// Pulses HOME and waits for the configured home-position feedback.
// Loss of bReady returns the FB to Idle without confirming completion.

FUNCTION_BLOCK FB_FanucHoming

VAR_INPUT
	bStart			: BOOL; // Rising edge starts homing while Idle and bReady; FALSE clears the FB error.
	bReady			: BOOL; // Enable permissive from FB_FanucEnable; must remain TRUE throughout the sequence.
	tHomingTimeout	: TIME := T#30S; // Maximum wait for bAt_Home = TRUE after the HOME pulse completes.
	stStatus		: ST_FanucStatus; // Live robot-status signals from FB_FanucStatus.
END_VAR

VAR_IN_OUT
	stControl	: ST_FanucControl; // Shared FANUC control structure; this FB writes Home only.
END_VAR

VAR_OUTPUT
	bBusy	: BOOL; // TRUE while in RequestHome or WaitComplete.
	bDone	: BOOL; // TRUE for one PLC scan when bAt_Home is TRUE in WaitComplete.
	bError	: BOOL; // TRUE in Error after a homing timeout or invalid state; cleared by bStart = FALSE.
	eState	: E_FanucHomingState; // Current state exposed for diagnostics and HMI.
END_VAR

VAR
	eCurrentState		: E_FanucHomingState := E_FanucHomingState.Idle; // Internal state used by the sequence.
	rtStart				: R_TRIG; // Detects the FALSE-to-TRUE transition of bStart.
	tonHomePulse		: TON; // Measures the HOME pulse duration in RequestHome.
	tonHomingTimeout	: TON; // Measures the wait for bAt_Home = TRUE in WaitComplete.
END_VAR

VAR CONSTANT
	tHomePulse	: TIME := T#200MS; // Requested duration of the HOME output pulse on UI[7].
END_VAR

(*
    FB_FanucHoming

    Purpose
    -------
    Controls the FANUC homing sequence and generates the HOME (UI[7])
    command used to trigger the configured homing macro or program.


    Homing sequence
    ---------------

        Idle
          |
          | bStart rising edge
          | + bReady
          v
        RequestHome
          |
          | HOME asserted for tHomePulse
          v
        WaitComplete
          |
          | bAt_Home = TRUE
          v
        Done
          |
          | one PLC scan
          v
        Idle


    Start behavior
    --------------
    bStart is treated as a momentary command.

    The R_TRIG detects the actual external FALSE -> TRUE transition:

        rtStart(CLK := bStart);

    The edge is accepted only when:

        bReady = TRUE
        AND
        eCurrentState = Idle

    A Start edge occurring while the robot is not Ready is ignored.

    If bStart goes TRUE before bReady becomes TRUE and remains TRUE,
    becoming Ready must NOT automatically start homing.

    bStart must first return FALSE and then receive a new rising edge.


    HOME pulse
    ----------
    RequestHome represents the HOME command pulse state.

    While RequestHome is active:

        stControl.Home = TRUE

    The HOME signal remains asserted for:

        tHomePulse

    After the pulse completes, the FB transitions to WaitComplete.


    Homing completion
    -----------------
    While in WaitComplete, the FB waits for:

        stStatus.bAt_Home = TRUE

    Once confirmed, the FB transitions to Done.

    bDone is TRUE for one PLC scan before the state returns to Idle.


    Ready interlock
    ---------------
    Homing may only start while:

        bReady = TRUE

    If bReady becomes FALSE during RequestHome or WaitComplete,
    the FB stops considering the homing sequence valid and returns
    to Idle.

    Returning this FB to Idle does not necessarily cancel a FANUC
    program or macro that has already started. Actual robot stopping
    behavior is controlled by the FANUC controller and its other UOP
    control inputs.


    Timeout
    -------
    While in WaitComplete, tonHomingTimeout runs for:

        tHomingTimeout

    If bAt_Home is not confirmed before the timeout expires,
    the FB transitions to Error.


    Error reset
    -----------
    To leave Error:

        bStart := FALSE

    The FB then returns to Idle.

    A new FALSE -> TRUE edge of bStart is required before another
    homing sequence can begin.


    FANUC prerequisites
    -------------------
    - HOME (UI[7]) must be configured to trigger the required
      homing macro or program.

    - stStatus.bAt_Home must represent the FANUC home-position
      feedback used by the application.


    Usage
    -----
    - Call this FB every PLC cycle.

    - Wire bReady from:

          FB_FanucEnable.bReady

    - Pass the same stControl instance used by the other FANUC
      command FBs and by FB_FanucControl.

    - Generate a rising edge on bStart to request homing.

    - Monitor:

          bBusy
          bDone
          bError
          eState
*)

// Start edge detection
// ============================================================================
//
// Detect the real external FALSE -> TRUE transition.
// Do not gate R_TRIG with bReady.
//
rtStart(CLK := bStart);

// State machine
// ============================================================================

CASE eCurrentState OF

    // IDLE ====================================================================
    E_FanucHomingState.Idle:

        // Accept Home only if the rising edge occurs while robot is Ready.
        IF rtStart.Q AND bReady THEN
            eCurrentState := E_FanucHomingState.RequestHome;
        END_IF;


    // REQUEST HOME ============================================================
    E_FanucHomingState.RequestHome:

        // Abort this FB sequence if robot Ready is lost.
        IF NOT bReady THEN
            eCurrentState := E_FanucHomingState.Idle;
        // HOME pulse completed.
        ELSIF tonHomePulse.Q THEN
            eCurrentState := E_FanucHomingState.WaitComplete;
        END_IF;

    // WAIT FOR HOME ===========================================================
    E_FanucHomingState.WaitComplete:

        IF NOT bReady THEN
            eCurrentState := E_FanucHomingState.Idle;
        // FANUC confirms Home position.
        ELSIF stStatus.bAt_Home THEN
            eCurrentState := E_FanucHomingState.Done;
        // Homing did not complete in time.
        ELSIF tonHomingTimeout.Q THEN
            eCurrentState := E_FanucHomingState.Error;
        END_IF;


    // DONE ====================================================================
    E_FanucHomingState.Done:

        // Done is exposed for one PLC scan.
        eCurrentState := E_FanucHomingState.Idle;

    // ERROR ===================================================================
    E_FanucHomingState.Error:

        // Require Start to be released before allowing another attempt.
        IF NOT bStart THEN
            eCurrentState := E_FanucHomingState.Idle;
        END_IF;

    // INVALID / UNKNOWN STATE =================================================
    ELSE
        eCurrentState := E_FanucHomingState.Error;
END_CASE;


// Timers
// ============================================================================
//
// Timers are enabled only by their corresponding state.

tonHomePulse(
    IN := (eCurrentState = E_FanucHomingState.RequestHome),
    PT := tHomePulse
);

tonHomingTimeout(
    IN := (eCurrentState = E_FanucHomingState.WaitComplete),
    PT := tHomingTimeout
);


// Derived FANUC control output
// ============================================================================
//
// HOME is asserted only during RequestHome and drops as soon as the
// configured pulse time has elapsed.

stControl.Home := (eCurrentState = E_FanucHomingState.RequestHome) AND NOT tonHomePulse.Q;

// Diagnostic outputs
// ============================================================================

eState := eCurrentState;

bBusy := (eCurrentState = E_FanucHomingState.RequestHome) OR (eCurrentState = E_FanucHomingState.WaitComplete);

bDone := (eCurrentState = E_FanucHomingState.Done);

bError := (eCurrentState = E_FanucHomingState.Error);

END_FUNCTION_BLOCK

(* stored: Version 1.1.0.1
   POU FB_FanucHoming: Id {d5b90ddc-612f-021f-8e89-4af80ef73b07}, SpecialFunc None *)
